FUNCTION_BLOCK PropertyObserver EXTENDS Object IMPLEMENTS I_Observer
VAR_INPUT
END_VAR
VAR_OUTPUT
END_VAR
VAR
    _name : STRING;
    _counter : INT;
END_VAR

METHOD Equals : BOOL
VAR_INPUT
    other : I_Equatable;
END_VAR
IF GetCounter() = GVL.CastHelper.I_EquatableToPropertyObserver(other)^.GetCounter() THEN
    Equals := TRUE;
ELSE
    Equals := FALSE;
END_IF
END_METHOD

METHOD GetCounter : INT
VAR_INPUT
END_VAR
GetCounter := _counter;
END_METHOD

METHOD OnError
_counter := _counter - 1;
END_METHOD

METHOD OnUpdate
_counter := _counter + 1;
END_METHOD

METHOD SetCounter
VAR_INPUT
    counter : INT;
END_VAR
_counter := counter;
END_METHOD

END_FUNCTION_BLOCK

(* stored: Version 1.1.0.1, ProductVersion 3.1.4024.6
   POU PropertyObserver: Id {4ee90097-ced5-48cf-a214-6cb507ca68bd}, SpecialFunc None
   Method Equals: Id {0942c81d-1b19-44f1-9932-d56d4230c531}
   Method GetCounter: Id {344ee8b2-6fbf-4e4f-ac4c-aba3e0b47456}
   Method OnError: Id {dcfdad8f-5616-4c87-b4ca-66d436821b42}
   Method OnUpdate: Id {43519026-10e7-428b-93a2-baf4968a1715}
   Method SetCounter: Id {f3f56185-b501-4574-889d-19524cdab58d} *)
